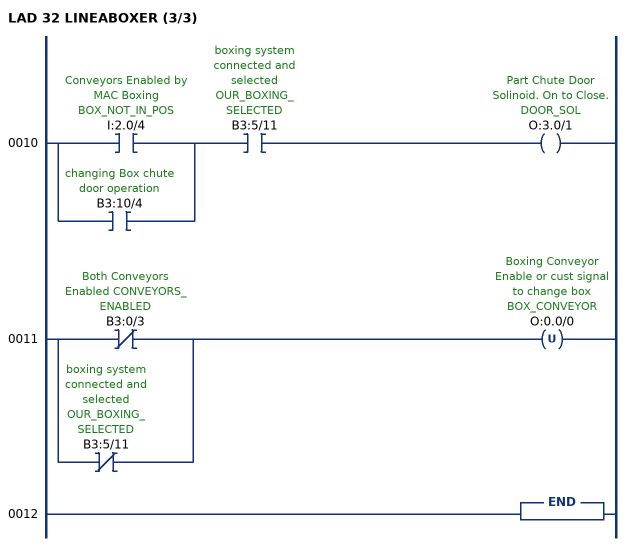
% Rung: 10 %
SOR BST XIC I:2.0/4 NXB XIC B3:10/4 BND XIC B3:5/11 OTE O:3.0/1 EOR
%   I:2.0/4  BOX_NOT_IN_POS  "Conveyors Enabled by MAC Boxing" %
%   B3:10/4  "changing Box chute door operation" %
%   B3:5/11  OUR_BOXING_SELECTED  "boxing system connected and selected" %
%   O:3.0/1  DOOR_SOL  "Part Chute Door Solinoid. On to Close." %
% Rung: 11 %
SOR BST XIO B3:0/3 NXB XIO B3:5/11 BND OTU O:0.0/0 EOR
%   B3:0/3  CONVEYORS_ENABLED  "Both Conveyors Enabled" %
%   B3:5/11  OUR_BOXING_SELECTED  "boxing system connected and selected" %
%   O:0.0/0  BOX_CONVEYOR  "Boxing Conveyor Enable or cust signal to change box" %
% Rung: 12 %
SOR END EOR

LADDER 33 "BULKBOXER"
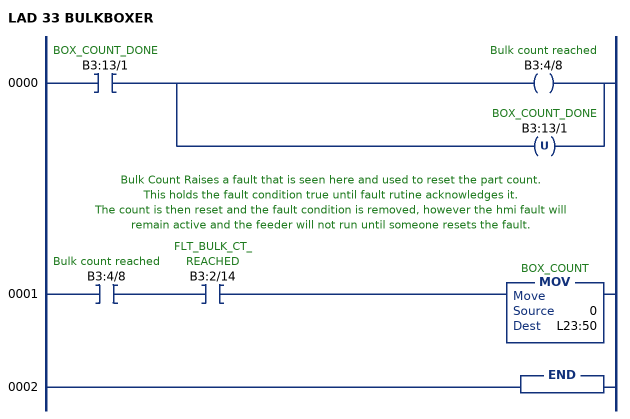
% Rung: 0 %
SOR XIC B3:13/1 BST OTE B3:4/8 NXB OTU B3:13/1 BND EOR
%   B3:13/1  BOX_COUNT_DONE %
%   B3:4/8  "Bulk count reached" %
% Rung: 1 %
% Bulk Count Raises a fault that is seen here and used to reset the part count.
% This holds the fault condition true until fault rutine acknowledges it.
% The count is then reset and the fault condition is removed, however the hmi fault will remain active and the feeder will not run until someone resets the fault. %
SOR XIC B3:4/8 XIC B3:2/14 MOV 0 L23:50 EOR
%   B3:4/8  "Bulk count reached" %
%   B3:2/14  FLT_BULK_CT_REACHED %
%   L23:50  BOX_COUNT %
% Rung: 2 %
SOR END EOR

LADDER 34 "CUSTBOXER"
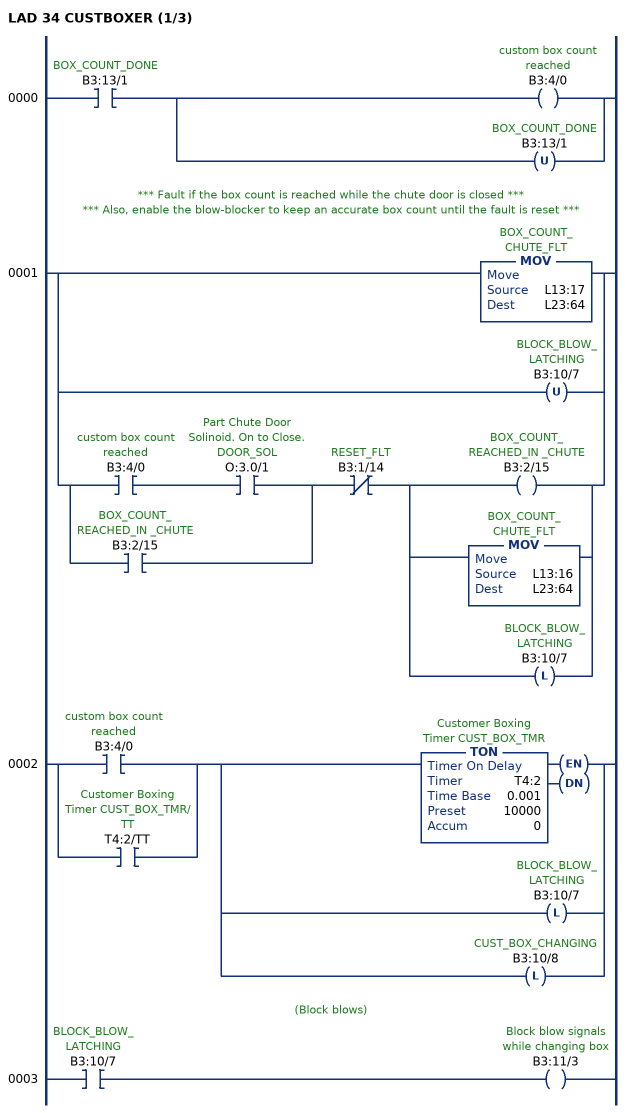
% Rung: 0 %
SOR XIC B3:13/1 BST OTE B3:4/0 NXB OTU B3:13/1 BND EOR
%   B3:13/1  BOX_COUNT_DONE %
%   B3:4/0  "custom box count reached" %
% Rung: 1 %
% *** Fault if the box count is reached while the chute door is closed ***
% *** Also, enable the blow-blocker to keep an accurate box count until the fault is reset *** %
SOR BST BST MOV L13:17 L23:64 NXB OTU B3:10/7 BND NXB BST XIC B3:4/0 XIC O:3.0/1 NXB XIC B3:2/15 BND XIO B3:1/14 BST OTE B3:2/15 NXB MOV L13:16 L23:64 NXB OTL B3:10/7 BND BND EOR
%   L13:17  FALSE %
%   L23:64  BOX_COUNT_CHUTE_FLT %
%   B3:10/7  BLOCK_BLOW_LATCHING %
%   B3:4/0  "custom box count reached" %
%   O:3.0/1  DOOR_SOL  "Part Chute Door Solinoid. On to Close." %
%   B3:2/15  "BOX_COUNT_REACHED_IN _CHUTE" %
%   B3:1/14  RESET_FLT %
%   L13:16  TRUE  "ONE TIME ENABLE FOR THE TIMES WHEN WE FORGET TO RE-ENABLE AFTER SHIPMENT" %
% Rung: 2 %
SOR BST XIC B3:4/0 NXB XIC T4:2/TT BND BST TON T4:2 0.001 10000 0 NXB OTL B3:10/7 NXB OTL B3:10/8 BND EOR
%   B3:4/0  "custom box count reached" %
%   T4:2  CUST_BOX_TMR  "Customer Boxing Timer" %
%   B3:10/7  BLOCK_BLOW_LATCHING %
%   B3:10/8  CUST_BOX_CHANGING %
% Rung: 3 %
% (Block blows) %
SOR XIC B3:10/7 OTE B3:11/3 EOR
%   B3:10/7  BLOCK_BLOW_LATCHING %
%   B3:11/3  "Block blow signals while changing box" %

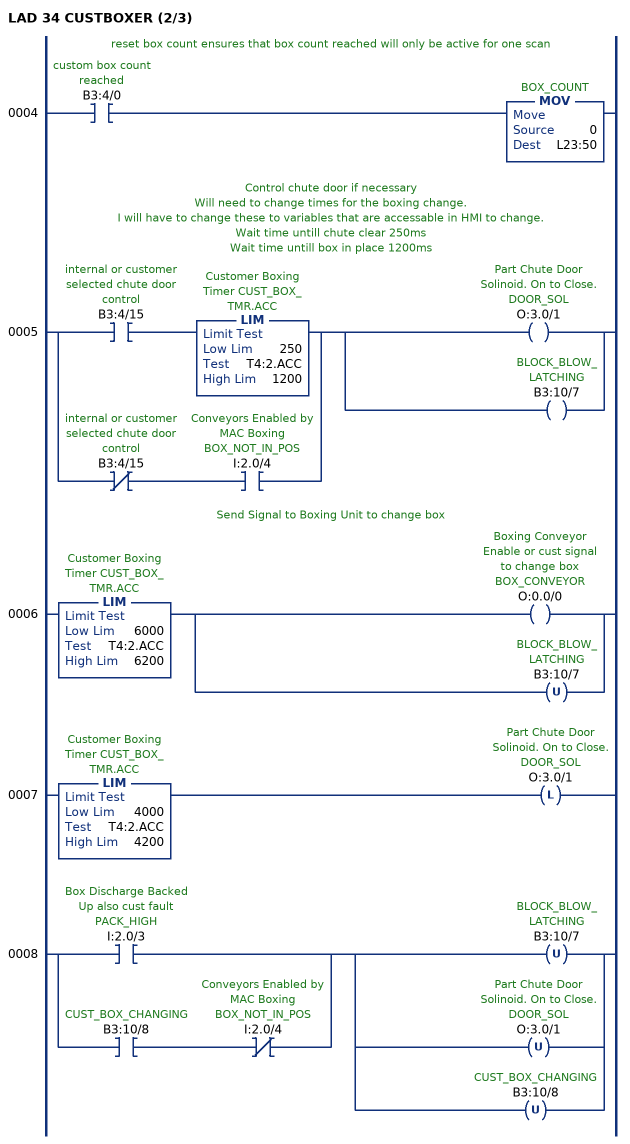
% Rung: 4 %
% reset box count ensures that box count reached will only be active for one scan %
SOR XIC B3:4/0 MOV 0 L23:50 EOR
%   B3:4/0  "custom box count reached" %
%   L23:50  BOX_COUNT %
% Rung: 5 %
% Control chute door if necessary
% 
% Will need to change times for the boxing change.
% I will have to change these to variables that are accessable in HMI to change.
% 
% Wait time untill chute clear 250ms
% Wait time untill box in place 1200ms %
SOR BST XIC B3:4/15 LIM 250 T4:2.ACC 1200 NXB XIO B3:4/15 XIC I:2.0/4 BND BST OTE O:3.0/1 NXB OTE B3:10/7 BND EOR
%   B3:4/15  "internal or customer selected chute door control" %
%   T4:2  CUST_BOX_TMR  "Customer Boxing Timer" %
%   I:2.0/4  BOX_NOT_IN_POS  "Conveyors Enabled by MAC Boxing" %
%   O:3.0/1  DOOR_SOL  "Part Chute Door Solinoid. On to Close." %
%   B3:10/7  BLOCK_BLOW_LATCHING %
% Rung: 6 %
% Send Signal to Boxing Unit to change box %
SOR LIM 6000 T4:2.ACC 6200 BST OTE O:0.0/0 NXB OTU B3:10/7 BND EOR
%   T4:2  CUST_BOX_TMR  "Customer Boxing Timer" %
%   O:0.0/0  BOX_CONVEYOR  "Boxing Conveyor Enable or cust signal to change box" %
%   B3:10/7  BLOCK_BLOW_LATCHING %
% Rung: 7 %
SOR LIM 4000 T4:2.ACC 4200 OTL O:3.0/1 EOR
%   T4:2  CUST_BOX_TMR  "Customer Boxing Timer" %
%   O:3.0/1  DOOR_SOL  "Part Chute Door Solinoid. On to Close." %
% Rung: 8 %
SOR BST XIC I:2.0/3 NXB XIC B3:10/8 XIO I:2.0/4 BND BST OTU B3:10/7 NXB OTU O:3.0/1 NXB OTU B3:10/8 BND EOR
%   I:2.0/3  PACK_HIGH  "Box Discharge Backed Up also cust fault" %
%   B3:10/8  CUST_BOX_CHANGING %
%   I:2.0/4  BOX_NOT_IN_POS  "Conveyors Enabled by MAC Boxing" %
%   B3:10/7  BLOCK_BLOW_LATCHING %
%   O:3.0/1  DOOR_SOL  "Part Chute Door Solinoid. On to Close." %

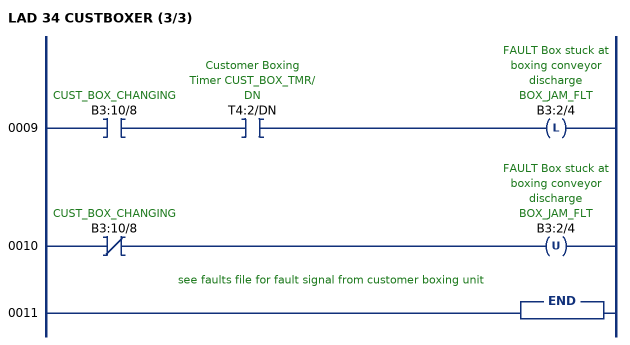
% Rung: 9 %
SOR XIC B3:10/8 XIC T4:2/DN OTL B3:2/4 EOR
%   B3:10/8  CUST_BOX_CHANGING %
%   T4:2  CUST_BOX_TMR  "Customer Boxing Timer" %
%   B3:2/4  BOX_JAM_FLT  "FAULT Box stuck at boxing conveyor discharge" %
% Rung: 10 %
SOR XIO B3:10/8 OTU B3:2/4 EOR
%   B3:10/8  CUST_BOX_CHANGING %
%   B3:2/4  BOX_JAM_FLT  "FAULT Box stuck at boxing conveyor discharge" %
% Rung: 11 %
% see faults file for fault signal from customer boxing unit %
SOR END EOR

LADDER 35 "CLEANUP"
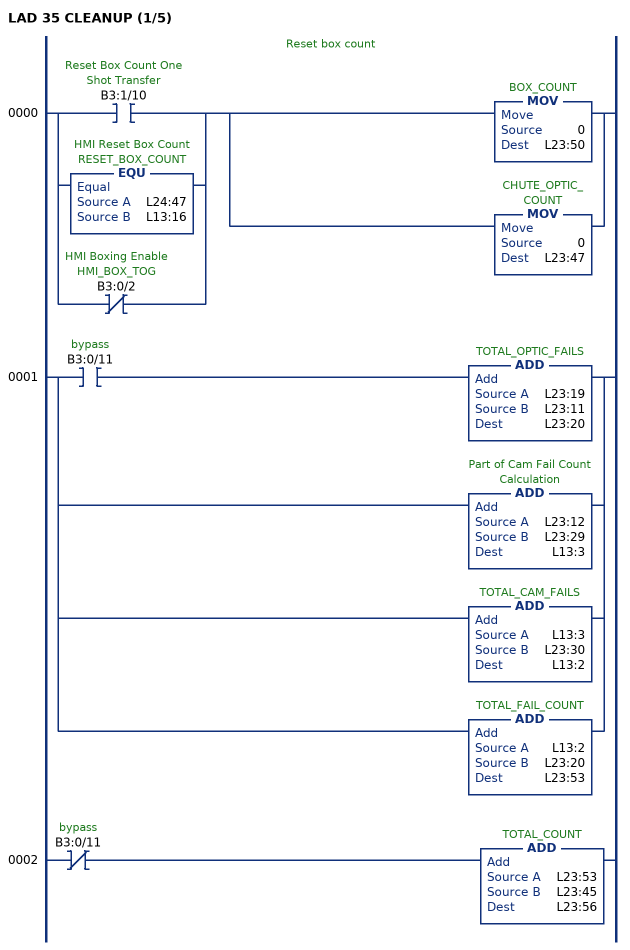
% Rung: 0 %
% Reset box count %
SOR BST XIC B3:1/10 NXB EQU L24:47 L13:16 NXB XIO B3:0/2 BND BST MOV 0 L23:50 NXB MOV 0 L23:47 BND EOR
%   B3:1/10  "Reset Box Count One Shot Transfer" %
%   L24:47  RESET_BOX_COUNT  "HMI Reset Box Count" %
%   L13:16  TRUE  "ONE TIME ENABLE FOR THE TIMES WHEN WE FORGET TO RE-ENABLE AFTER SHIPMENT" %
%   B3:0/2  HMI_BOX_TOG  "HMI Boxing Enable" %
%   L23:50  BOX_COUNT %
%   L23:47  CHUTE_OPTIC_COUNT %
% Rung: 1 %
SOR BST XIC B3:0/11 ADD L23:19 L23:11 L23:20 NXB ADD L23:12 L23:29 L13:3 NXB ADD L13:3 L23:30 L13:2 NXB ADD L13:2 L23:20 L23:53 BND EOR
%   B3:0/11  "bypass" %
%   L23:19  TOP_OPT_FAIL_CT %
%   L23:11  BOT_OPT_FAIL_CT %
%   L23:20  TOTAL_OPTIC_FAILS %
%   L23:12  BOT_NON_PASS  "parts missed BOT camera" %
%   L23:29  SIDE_NON_PASS  "parts missed side camera" %
%   L13:3  "Part of Cam Fail Count Calculation" %
%   L23:30  TOP_NON_PASS  "Parts Missed Top Camera" %
%   L13:2  TOTAL_CAM_FAILS %
%   L23:53  TOTAL_FAIL_COUNT %
% Rung: 2 %
SOR XIO B3:0/11 ADD L23:53 L23:45 L23:56 EOR
%   B3:0/11  "bypass" %
%   L23:53  TOTAL_FAIL_COUNT %
%   L23:45  BLOW_COUNT %
%   L23:56  TOTAL_COUNT %

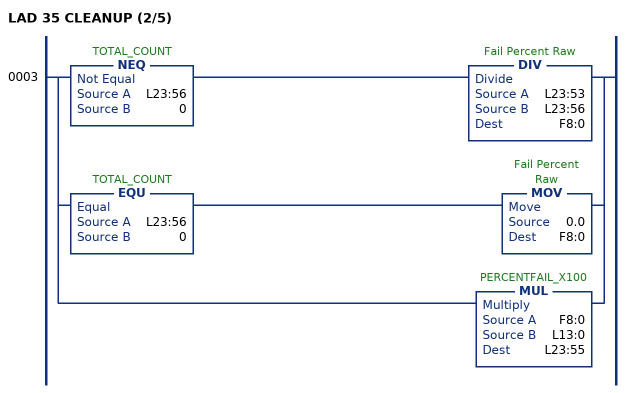
% Rung: 3 %
SOR BST NEQ L23:56 0 DIV L23:53 L23:56 F8:0 NXB EQU L23:56 0 MOV 0.0 F8:0 NXB MUL F8:0 L13:0 L23:55 BND EOR
%   L23:56  TOTAL_COUNT %
%   L23:53  TOTAL_FAIL_COUNT %
%   F8:0  "Fail Percent Raw" %
%   L13:0  "multiplyer to translate percent" %
%   L23:55  PERCENTFAIL_X100 %

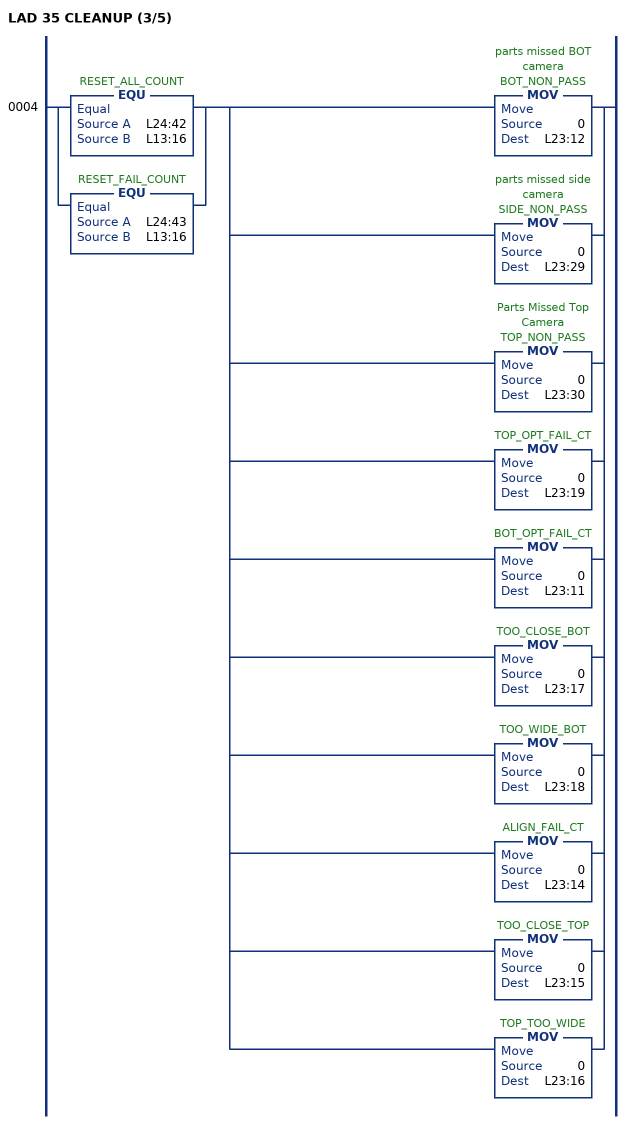
% Rung: 4 %
SOR BST EQU L24:42 L13:16 NXB EQU L24:43 L13:16 BND BST MOV 0 L23:12 NXB MOV 0 L23:29 NXB MOV 0 L23:30 NXB MOV 0 L23:19 NXB MOV 0 L23:11 NXB MOV 0 L23:17 NXB MOV 0 L23:18 NXB MOV 0 L23:14 NXB MOV 0 L23:15 NXB MOV 0 L23:16 BND EOR
%   L24:42  RESET_ALL_COUNT %
%   L13:16  TRUE  "ONE TIME ENABLE FOR THE TIMES WHEN WE FORGET TO RE-ENABLE AFTER SHIPMENT" %
%   L24:43  RESET_FAIL_COUNT %
%   L23:12  BOT_NON_PASS  "parts missed BOT camera" %
%   L23:29  SIDE_NON_PASS  "parts missed side camera" %
%   L23:30  TOP_NON_PASS  "Parts Missed Top Camera" %
%   L23:19  TOP_OPT_FAIL_CT %
%   L23:11  BOT_OPT_FAIL_CT %
%   L23:17  TOO_CLOSE_BOT %
%   L23:18  TOO_WIDE_BOT %
%   L23:14  ALIGN_FAIL_CT %
%   L23:15  TOO_CLOSE_TOP %
%   L23:16  TOP_TOO_WIDE %

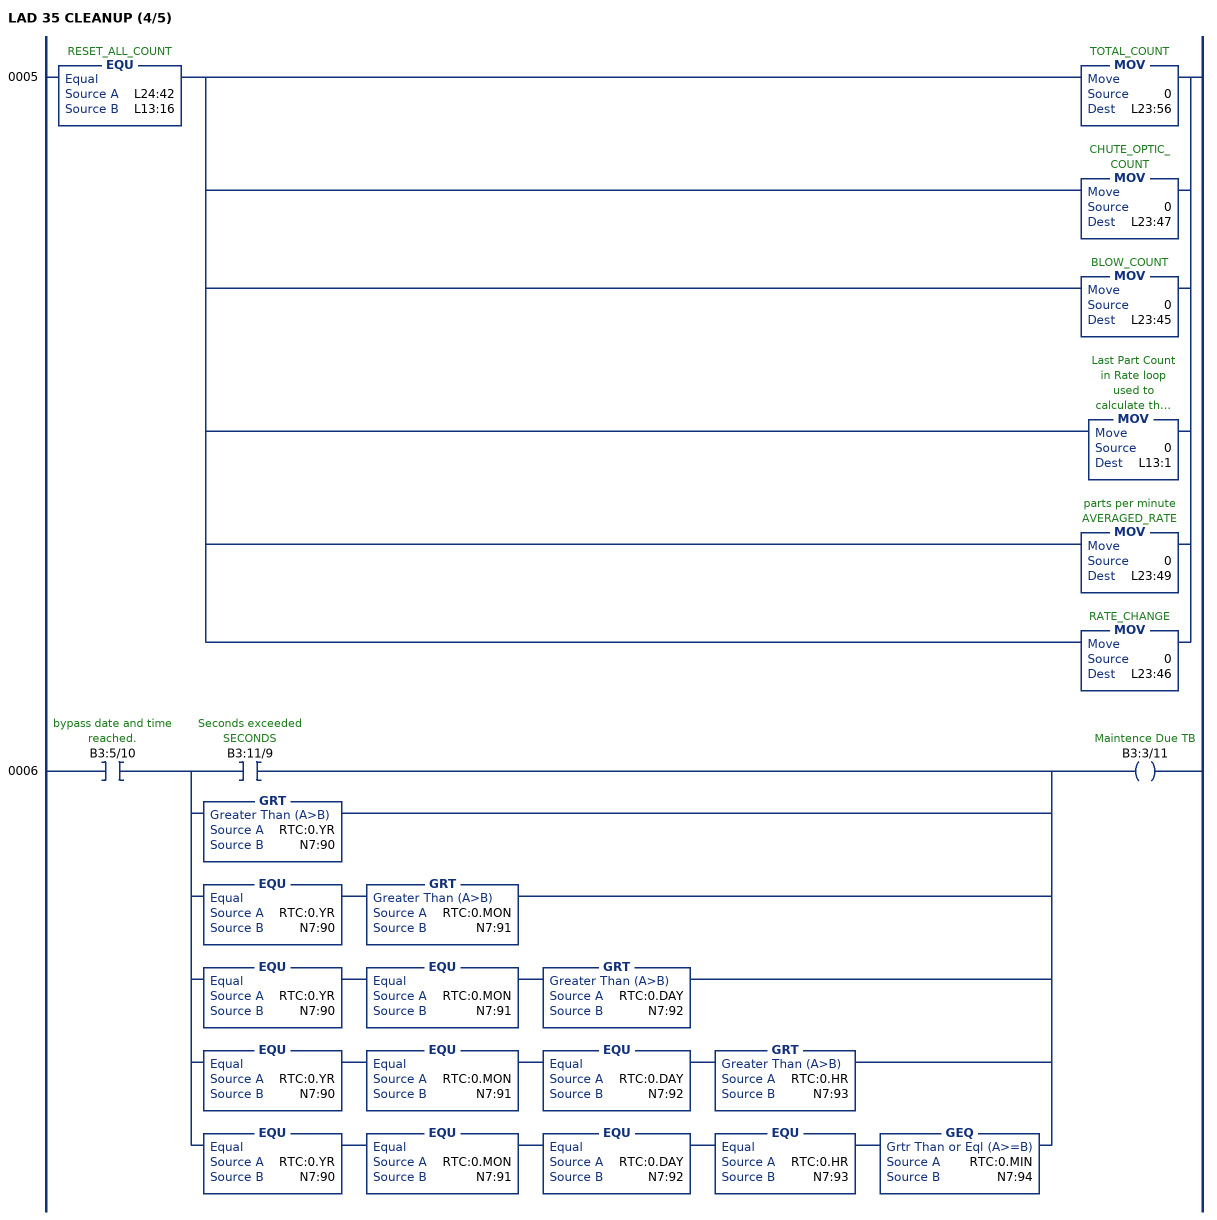
% Rung: 5 %
SOR EQU L24:42 L13:16 BST MOV 0 L23:56 NXB MOV 0 L23:47 NXB MOV 0 L23:45 NXB MOV 0 L13:1 NXB MOV 0 L23:49 NXB MOV 0 L23:46 BND EOR
%   L24:42  RESET_ALL_COUNT %
%   L13:16  TRUE  "ONE TIME ENABLE FOR THE TIMES WHEN WE FORGET TO RE-ENABLE AFTER SHIPMENT" %
%   L23:56  TOTAL_COUNT %
%   L23:47  CHUTE_OPTIC_COUNT %
%   L23:45  BLOW_COUNT %
%   L13:1  "Last Part Count in Rate loop used to calculate the last cycle part count" %
%   L23:49  AVERAGED_RATE  "parts per minute" %
%   L23:46  RATE_CHANGE %
% Rung: 6 %
SOR XIC B3:5/10 BST XIC B3:11/9 NXB GRT RTC:0.YR N7:90 NXB EQU RTC:0.YR N7:90 GRT RTC:0.MON N7:91 NXB EQU RTC:0.YR N7:90 EQU RTC:0.MON N7:91 GRT RTC:0.DAY N7:92 NXB EQU RTC:0.YR N7:90 EQU RTC:0.MON N7:91 EQU RTC:0.DAY N7:92 GRT RTC:0.HR N7:93 NXB EQU RTC:0.YR N7:90 EQU RTC:0.MON N7:91 EQU RTC:0.DAY N7:92 EQU RTC:0.HR N7:93 GEQ RTC:0.MIN N7:94 BND OTE B3:3/11 EOR
%   B3:5/10  "bypass date and time reached." %
%   B3:11/9  SECONDS  "Seconds exceeded" %
%   N7:90  RTC %
%   B3:3/11  TB  "Maintence Due" %

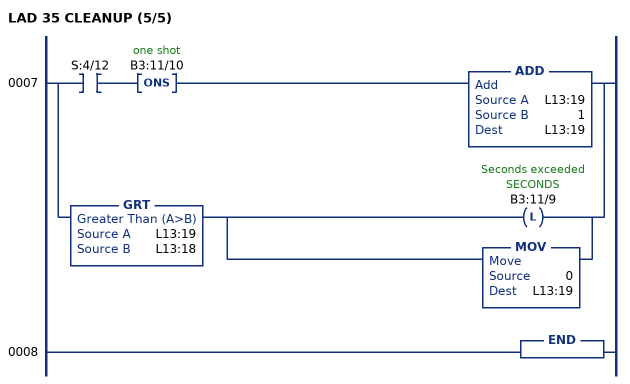
% Rung: 7 %
SOR BST XIC S:4/12 ONS B3:11/10 ADD L13:19 1 L13:19 NXB GRT L13:19 L13:18 BST OTL B3:11/9 NXB MOV 0 L13:19 BND BND EOR
%   B3:11/10  "one shot" %
%   L13:18  MAX %
%   B3:11/9  SECONDS  "Seconds exceeded" %
% Rung: 8 %
SOR END EOR

LADDER 36 "J_CUST_BOX"    % Justin's customer boxing ladder %
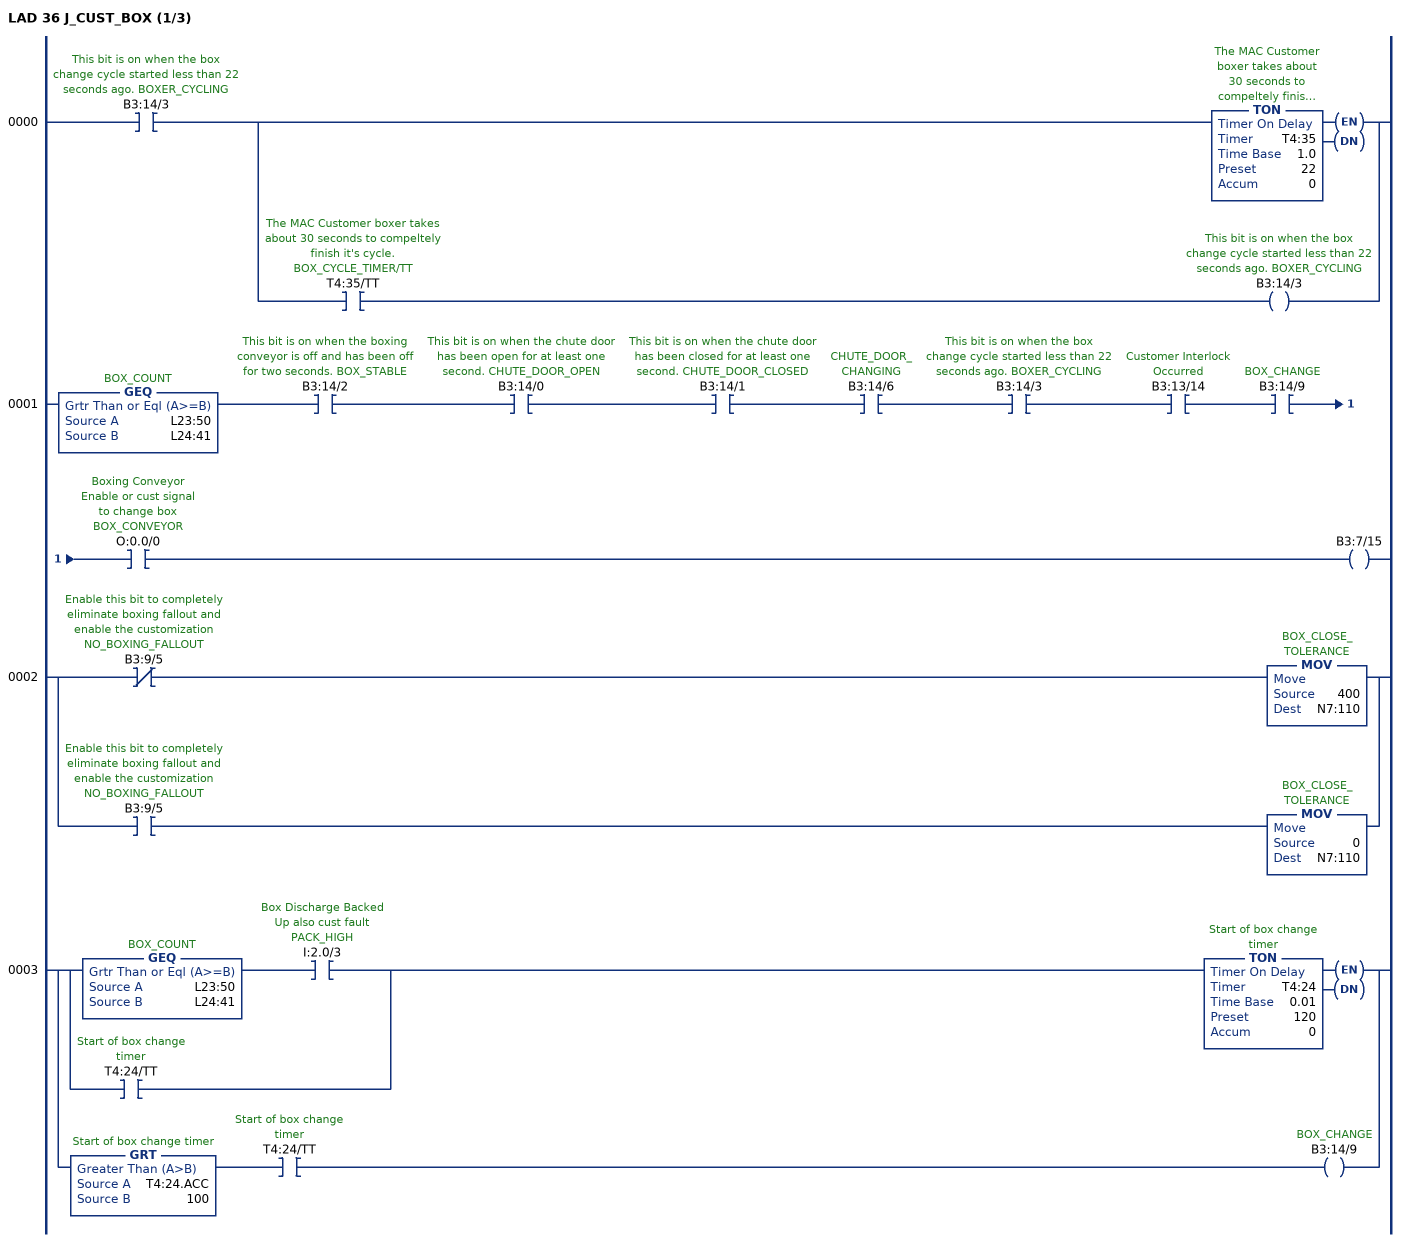
% Rung: 0 %
SOR XIC B3:14/3 BST TON T4:35 1.0 22 0 NXB XIC T4:35/TT OTE B3:14/3 BND EOR
%   B3:14/3  BOXER_CYCLING  "This bit is on when the box change cycle started less than 22 seconds ago." %
%   T4:35  BOX_CYCLE_TIMER  "The MAC Customer boxer takes about 30 seconds to compeltely finish it's cycle." %
% Rung: 1 %
SOR GEQ L23:50 L24:41 XIC B3:14/2 XIC B3:14/0 XIC B3:14/1 XIC B3:14/6 XIC B3:14/3 XIC B3:13/14 XIC B3:14/9 XIC O:0.0/0 OTE B3:7/15 EOR
%   L23:50  BOX_COUNT %
%   L24:41  BOX_COUNT_LIMIT %
%   B3:14/2  BOX_STABLE  "This bit is on when the boxing conveyor is off and has been off for two seconds." %
%   B3:14/0  CHUTE_DOOR_OPEN  "This bit is on when the chute door has been open for at least one second." %
%   B3:14/1  CHUTE_DOOR_CLOSED  "This bit is on when the chute door has been closed for at least one second." %
%   B3:14/6  CHUTE_DOOR_CHANGING %
%   B3:14/3  BOXER_CYCLING  "This bit is on when the box change cycle started less than 22 seconds ago." %
%   B3:13/14  "Customer Interlock Occurred" %
%   B3:14/9  BOX_CHANGE %
%   O:0.0/0  BOX_CONVEYOR  "Boxing Conveyor Enable or cust signal to change box" %
% Rung: 2 %
SOR BST XIO B3:9/5 MOV 400 N7:110 NXB XIC B3:9/5 MOV 0 N7:110 BND EOR
%   B3:9/5  NO_BOXING_FALLOUT  "Enable this bit to completely eliminate boxing fallout and enable the customization" %
%   N7:110  BOX_CLOSE_TOLERANCE %
% Rung: 3 %
SOR BST BST GEQ L23:50 L24:41 XIC I:2.0/3 NXB XIC T4:24/TT BND TON T4:24 0.01 120 0 NXB GRT T4:24.ACC 100 XIC T4:24/TT OTE B3:14/9 BND EOR
%   L23:50  BOX_COUNT %
%   L24:41  BOX_COUNT_LIMIT %
%   I:2.0/3  PACK_HIGH  "Box Discharge Backed Up also cust fault" %
%   T4:24  "Start of box change timer" %
%   B3:14/9  BOX_CHANGE %

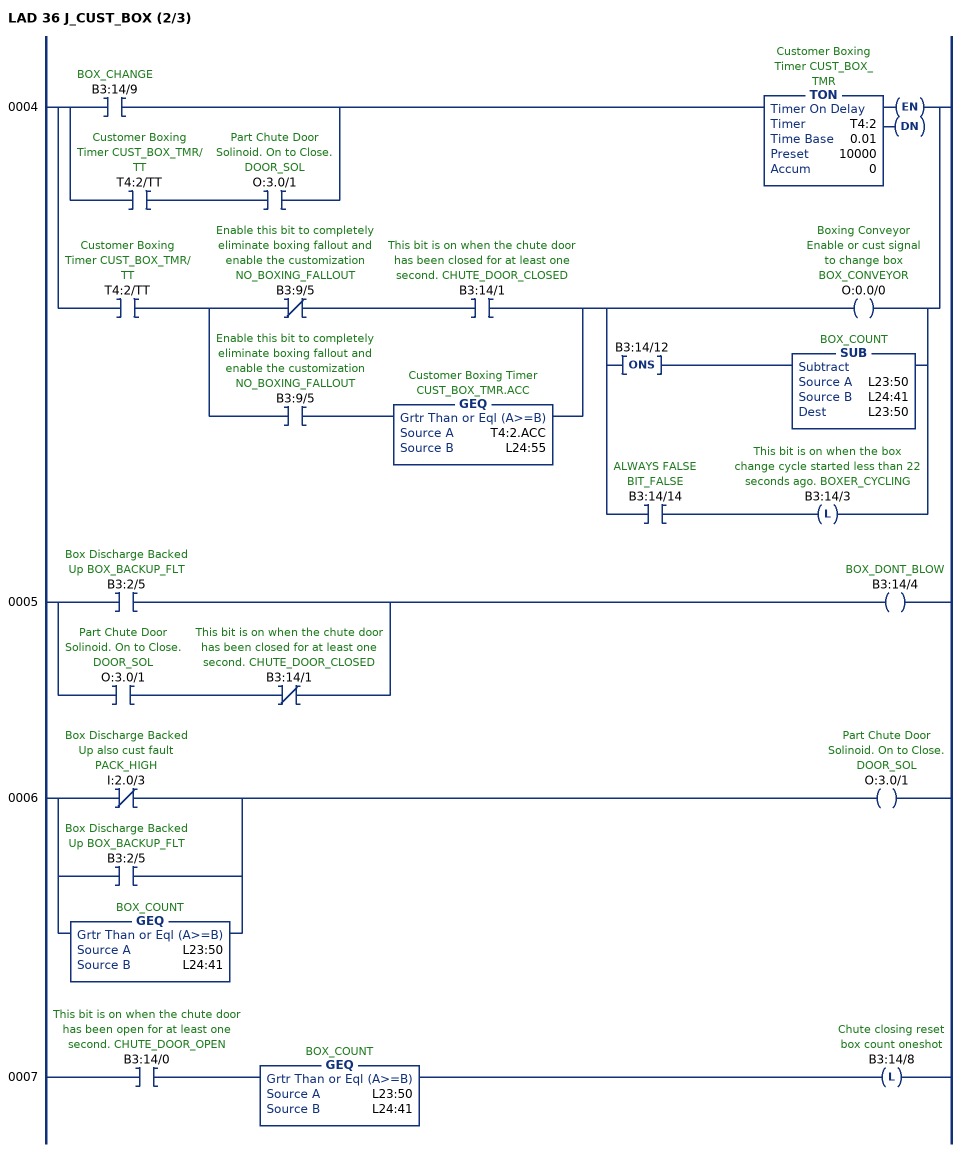
% Rung: 4 %
SOR BST BST XIC B3:14/9 NXB XIC T4:2/TT XIC O:3.0/1 BND TON T4:2 0.01 10000 0 NXB XIC T4:2/TT BST XIO B3:9/5 XIC B3:14/1 NXB XIC B3:9/5 GEQ T4:2.ACC L24:55 BND BST OTE O:0.0/0 NXB ONS B3:14/12 SUB L23:50 L24:41 L23:50 NXB XIC B3:14/14 OTL B3:14/3 BND BND EOR
%   B3:14/9  BOX_CHANGE %
%   T4:2  CUST_BOX_TMR  "Customer Boxing Timer" %
%   O:3.0/1  DOOR_SOL  "Part Chute Door Solinoid. On to Close." %
%   B3:9/5  NO_BOXING_FALLOUT  "Enable this bit to completely eliminate boxing fallout and enable the customization" %
%   B3:14/1  CHUTE_DOOR_CLOSED  "This bit is on when the chute door has been closed for at least one second." %
%   L24:55  CHUTE_CLOSE_DELAY  "Timer to allow parts to pass through the chute" %
%   O:0.0/0  BOX_CONVEYOR  "Boxing Conveyor Enable or cust signal to change box" %
%   L23:50  BOX_COUNT %
%   L24:41  BOX_COUNT_LIMIT %
%   B3:14/14  BIT_FALSE  "ALWAYS FALSE" %
%   B3:14/3  BOXER_CYCLING  "This bit is on when the box change cycle started less than 22 seconds ago." %
% Rung: 5 %
SOR BST XIC B3:2/5 NXB XIC O:3.0/1 XIO B3:14/1 BND OTE B3:14/4 EOR
%   B3:2/5  BOX_BACKUP_FLT  "Box Discharge Backed Up" %
%   O:3.0/1  DOOR_SOL  "Part Chute Door Solinoid. On to Close." %
%   B3:14/1  CHUTE_DOOR_CLOSED  "This bit is on when the chute door has been closed for at least one second." %
%   B3:14/4  BOX_DONT_BLOW %
% Rung: 6 %
SOR BST XIO I:2.0/3 NXB XIC B3:2/5 NXB GEQ L23:50 L24:41 BND OTE O:3.0/1 EOR
%   I:2.0/3  PACK_HIGH  "Box Discharge Backed Up also cust fault" %
%   B3:2/5  BOX_BACKUP_FLT  "Box Discharge Backed Up" %
%   L23:50  BOX_COUNT %
%   L24:41  BOX_COUNT_LIMIT %
%   O:3.0/1  DOOR_SOL  "Part Chute Door Solinoid. On to Close." %
% Rung: 7 %
SOR XIC B3:14/0 GEQ L23:50 L24:41 OTL B3:14/8 EOR
%   B3:14/0  CHUTE_DOOR_OPEN  "This bit is on when the chute door has been open for at least one second." %
%   L23:50  BOX_COUNT %
%   L24:41  BOX_COUNT_LIMIT %
%   B3:14/8  "Chute closing reset box count oneshot" %

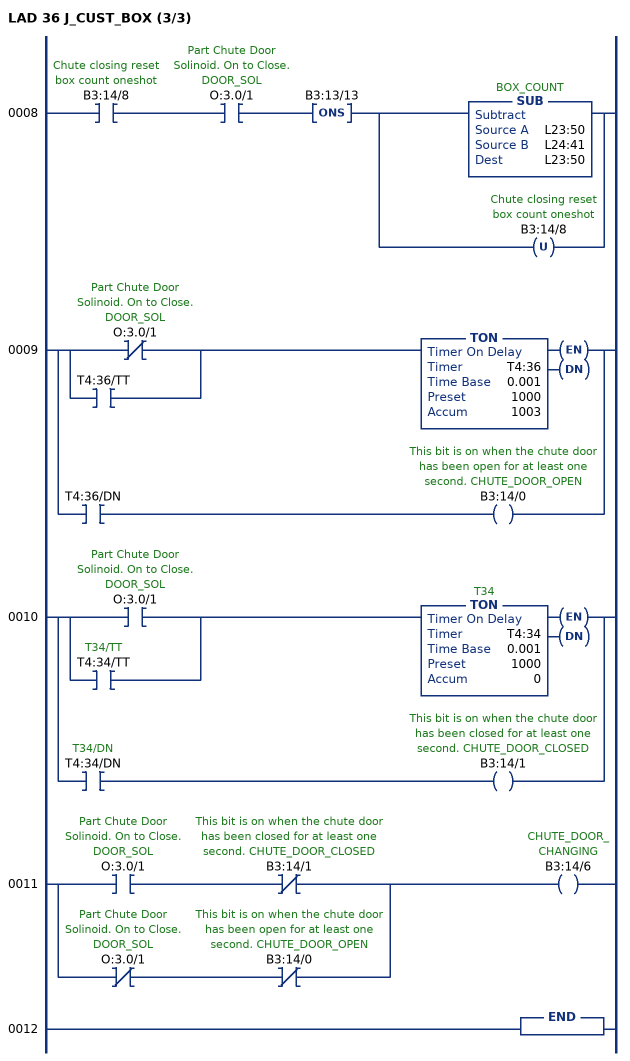
% Rung: 8 %
SOR XIC B3:14/8 XIC O:3.0/1 ONS B3:13/13 BST SUB L23:50 L24:41 L23:50 NXB OTU B3:14/8 BND EOR
%   B3:14/8  "Chute closing reset box count oneshot" %
%   O:3.0/1  DOOR_SOL  "Part Chute Door Solinoid. On to Close." %
%   L23:50  BOX_COUNT %
%   L24:41  BOX_COUNT_LIMIT %
% Rung: 9 %
SOR BST BST XIO O:3.0/1 NXB XIC T4:36/TT BND TON T4:36 0.001 1000 1003 NXB XIC T4:36/DN OTE B3:14/0 BND EOR
%   O:3.0/1  DOOR_SOL  "Part Chute Door Solinoid. On to Close." %
%   B3:14/0  CHUTE_DOOR_OPEN  "This bit is on when the chute door has been open for at least one second." %
% Rung: 10 %
SOR BST BST XIC O:3.0/1 NXB XIC T4:34/TT BND TON T4:34 0.001 1000 0 NXB XIC T4:34/DN OTE B3:14/1 BND EOR
%   O:3.0/1  DOOR_SOL  "Part Chute Door Solinoid. On to Close." %
%   T4:34  T34 %
%   B3:14/1  CHUTE_DOOR_CLOSED  "This bit is on when the chute door has been closed for at least one second." %
% Rung: 11 %
SOR BST XIC O:3.0/1 XIO B3:14/1 NXB XIO O:3.0/1 XIO B3:14/0 BND OTE B3:14/6 EOR
%   O:3.0/1  DOOR_SOL  "Part Chute Door Solinoid. On to Close." %
%   B3:14/1  CHUTE_DOOR_CLOSED  "This bit is on when the chute door has been closed for at least one second." %
%   B3:14/0  CHUTE_DOOR_OPEN  "This bit is on when the chute door has been open for at least one second." %
%   B3:14/6  CHUTE_DOOR_CHANGING %
% Rung: 12 %
SOR END EOR

LADDER 37 "BOXING"
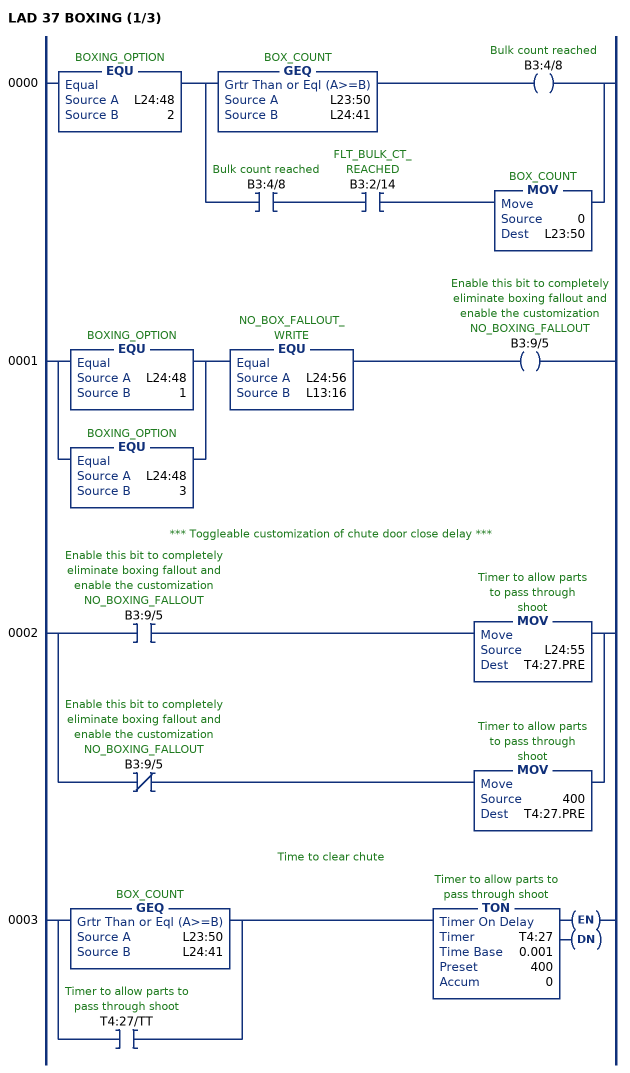
% Rung: 0 %
SOR EQU L24:48 2 BST GEQ L23:50 L24:41 OTE B3:4/8 NXB XIC B3:4/8 XIC B3:2/14 MOV 0 L23:50 BND EOR
%   L24:48  BOXING_OPTION %
%   L23:50  BOX_COUNT %
%   L24:41  BOX_COUNT_LIMIT %
%   B3:4/8  "Bulk count reached" %
%   B3:2/14  FLT_BULK_CT_REACHED %
% Rung: 1 %
SOR BST EQU L24:48 1 NXB EQU L24:48 3 BND EQU L24:56 L13:16 OTE B3:9/5 EOR
%   L24:48  BOXING_OPTION %
%   L24:56  NO_BOX_FALLOUT_WRITE %
%   L13:16  TRUE  "ONE TIME ENABLE FOR THE TIMES WHEN WE FORGET TO RE-ENABLE AFTER SHIPMENT" %
%   B3:9/5  NO_BOXING_FALLOUT  "Enable this bit to completely eliminate boxing fallout and enable the customization" %
% Rung: 2 %
% *** Toggleable customization of chute door close delay *** %
SOR BST XIC B3:9/5 MOV L24:55 T4:27.PRE NXB XIO B3:9/5 MOV 400 T4:27.PRE BND EOR
%   B3:9/5  NO_BOXING_FALLOUT  "Enable this bit to completely eliminate boxing fallout and enable the customization" %
%   L24:55  CHUTE_CLOSE_DELAY  "Timer to allow parts to pass through the chute" %
%   T4:27  "Timer to allow parts to pass through shoot" %
% Rung: 3 %
% Time to clear chute %
SOR BST GEQ L23:50 L24:41 NXB XIC T4:27/TT BND TON T4:27 0.001 400 0 EOR
%   L23:50  BOX_COUNT %
%   L24:41  BOX_COUNT_LIMIT %
%   T4:27  "Timer to allow parts to pass through shoot" %

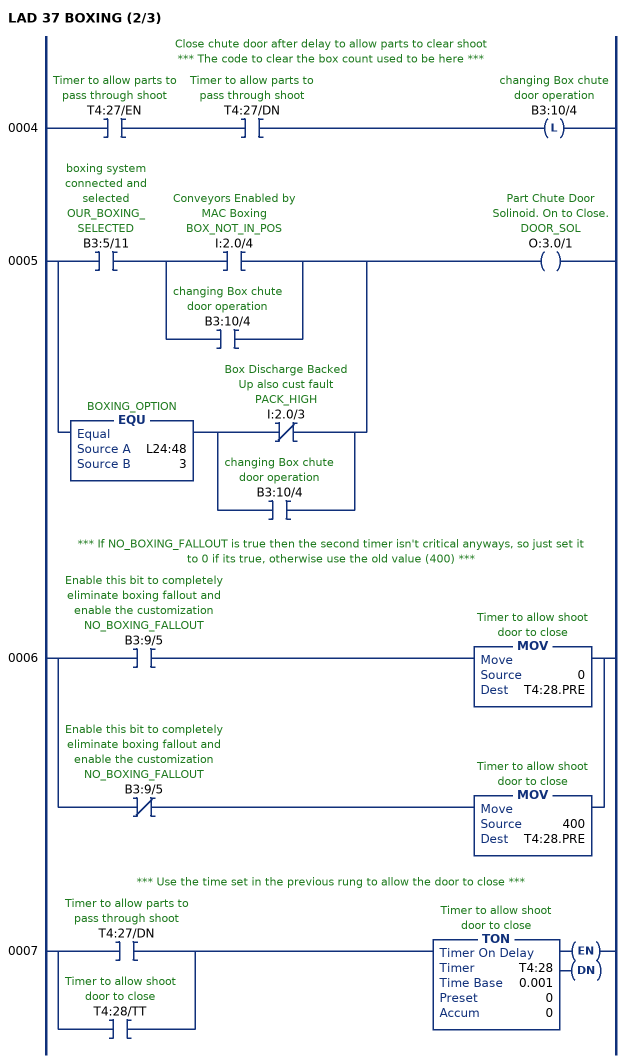
% Rung: 4 %
% Close chute door after delay to allow parts to clear shoot
% *** The code to clear the box count used to be here *** %
SOR XIC T4:27/EN XIC T4:27/DN OTL B3:10/4 EOR
%   T4:27  "Timer to allow parts to pass through shoot" %
%   B3:10/4  "changing Box chute door operation" %
% Rung: 5 %
SOR BST XIC B3:5/11 BST XIC I:2.0/4 NXB XIC B3:10/4 BND NXB EQU L24:48 3 BST XIO I:2.0/3 NXB XIC B3:10/4 BND BND OTE O:3.0/1 EOR
%   B3:5/11  OUR_BOXING_SELECTED  "boxing system connected and selected" %
%   I:2.0/4  BOX_NOT_IN_POS  "Conveyors Enabled by MAC Boxing" %
%   B3:10/4  "changing Box chute door operation" %
%   L24:48  BOXING_OPTION %
%   I:2.0/3  PACK_HIGH  "Box Discharge Backed Up also cust fault" %
%   O:3.0/1  DOOR_SOL  "Part Chute Door Solinoid. On to Close." %
% Rung: 6 %
% *** If NO_BOXING_FALLOUT is true then the second timer isn't critical anyways, so just set it to 0 if its true, otherwise use the old value (400) *** %
SOR BST XIC B3:9/5 MOV 0 T4:28.PRE NXB XIO B3:9/5 MOV 400 T4:28.PRE BND EOR
%   B3:9/5  NO_BOXING_FALLOUT  "Enable this bit to completely eliminate boxing fallout and enable the customization" %
%   T4:28  "Timer to allow shoot door to close" %
% Rung: 7 %
% *** Use the time set in the previous rung to allow the door to close *** %
SOR BST XIC T4:27/DN NXB XIC T4:28/TT BND TON T4:28 0.001 0 0 EOR
%   T4:27  "Timer to allow parts to pass through shoot" %
%   T4:28  "Timer to allow shoot door to close" %

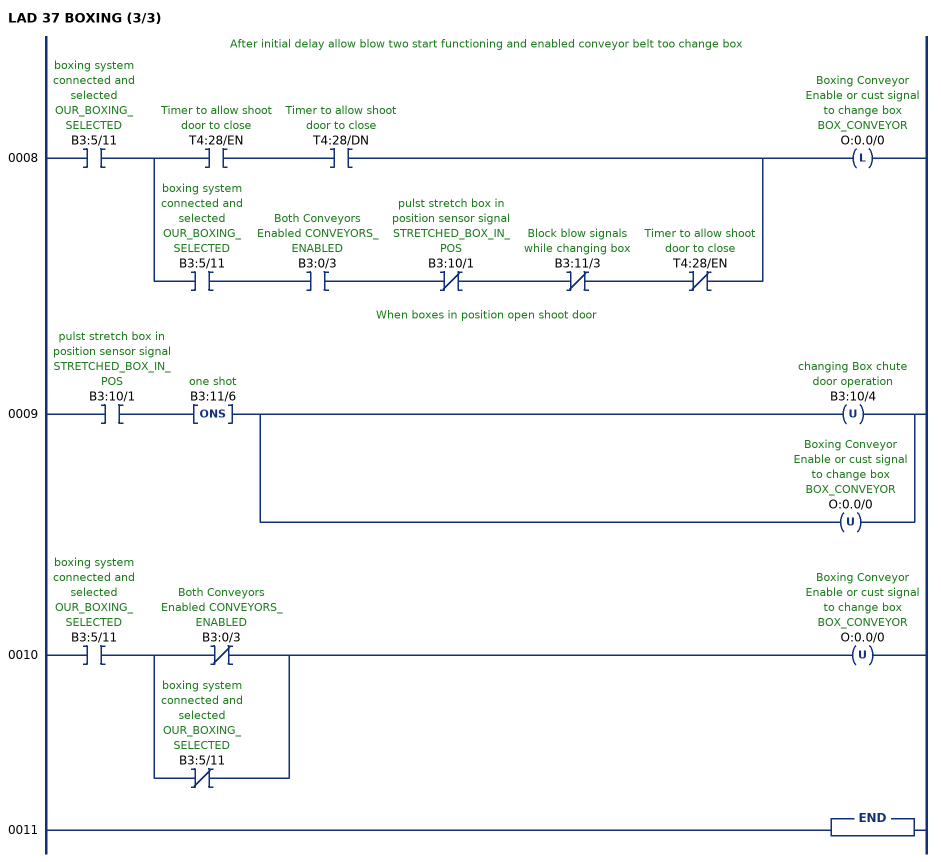
% Rung: 8 %
% After initial delay allow blow two start functioning and enabled conveyor belt too change box %
SOR XIC B3:5/11 BST XIC T4:28/EN XIC T4:28/DN NXB XIC B3:5/11 XIC B3:0/3 XIO B3:10/1 XIO B3:11/3 XIO T4:28/EN BND OTL O:0.0/0 EOR
%   B3:5/11  OUR_BOXING_SELECTED  "boxing system connected and selected" %
%   T4:28  "Timer to allow shoot door to close" %
%   B3:0/3  CONVEYORS_ENABLED  "Both Conveyors Enabled" %
%   B3:10/1  STRETCHED_BOX_IN_POS  "pulst stretch box in position sensor signal" %
%   B3:11/3  "Block blow signals while changing box" %
%   O:0.0/0  BOX_CONVEYOR  "Boxing Conveyor Enable or cust signal to change box" %
% Rung: 9 %
% When boxes in position open shoot door %
SOR XIC B3:10/1 ONS B3:11/6 BST OTU B3:10/4 NXB OTU O:0.0/0 BND EOR
%   B3:10/1  STRETCHED_BOX_IN_POS  "pulst stretch box in position sensor signal" %
%   B3:11/6  "one shot" %
%   B3:10/4  "changing Box chute door operation" %
%   O:0.0/0  BOX_CONVEYOR  "Boxing Conveyor Enable or cust signal to change box" %
% Rung: 10 %
SOR XIC B3:5/11 BST XIO B3:0/3 NXB XIO B3:5/11 BND OTU O:0.0/0 EOR
%   B3:5/11  OUR_BOXING_SELECTED  "boxing system connected and selected" %
%   B3:0/3  CONVEYORS_ENABLED  "Both Conveyors Enabled" %
%   O:0.0/0  BOX_CONVEYOR  "Boxing Conveyor Enable or cust signal to change box" %
% Rung: 11 %
SOR END EOR

OTHER DOCUMENTED ADDRESSES
  100000L  
  B3:2/12  "Rate Drop Fault Possible Feed Jam"
  B3:5/8  OFF
  B3:5/13  "bot result toggle"
  B3:6/5  "bottom top camra pass zone"
  B3:6/6  "one shot"
  B3:6/7  EI3_OLD  "Enable Inspection 3"
  B3:6/9  CONV_ON  "both conveyors enabled"
  B3:6/10  "Bypass un-needed code untill completed !!!!!!!!!!!!!!!!"
  B3:6/15  "nothing"
  B3:7/2  "bypass"
  B3:7/5  "extra bypass"
  B3:7/8  "top camera pass part zone"
  B3:7/11  "good part detected at top top"
  B3:7/12  "side camera pass part zone"
  B3:7/14  "passing part present bottom top camera"
  B3:8/0  "bypass extra trigger camera 1"
  B3:8/1  "bypass extra trigger camera 2"
  B3:8/2  "bypass extra trigger camera 3"
  B3:8/3  "bypass extra trigger camera 4"
  B3:8/5  TEST  "FORCE FEED ON/OFF"
  B3:8/6  "a bypass bit"
  B3:8/7  "a bypass bit"
  B3:8/11  ET4  "extra trigger camera 4"
  B3:8/12  "start bottom top camera responce"
  B3:8/13  "extra blow signal for testing"
  B3:8/15  "start side camera responce"
  B3:9/2  "one shot"
  B3:9/4  "start top camera responce"
  B3:9/7  "C1t"
  B3:9/8  "C2D"
  B3:9/9  "C2t"
  B3:9/14  "input from hmi to reset count"
  B3:10/0  "bypass part too close"
  B3:10/5  "one shot"
  B3:10/6  "excessive data output time"
  B3:10/9  "one shot"
  B3:10/10  "one shot"
  B3:10/14  "Dont use"
  B3:11/0  "bypass unused portion of code"
  B3:11/1  "bypass"
  B3:11/2  "Enable encoder belt movement simulation when testing"
  B3:11/7  "one shot"
  B3:11/11  "one shot"
  B3:11/13  TEST_TRIG_SIG
  B3:11/14  SOC  "start delay to false optic cycle"
  B3:11/15  "one shot"
  B3:12/2  "Command 2 Oneshot"
  B3:12/3  "Command 2 Active"
  B3:12/4  "Command3 Oneshot"
  B3:12/5  "Command 3 Active"
  B3:12/6  "Inspection Command Counter"
  B3:12/7  "Command 4 Active"
  B3:12/8  "Command 4 Oneshot"
  B3:12/15  "FALSE"
  B3:13/5  "bypass"
  B3:13/12  "Test Trigger to laser Spacing"
  B3:13/15  "Test Signals"
  B3:14  BOXING_STATUS  "Various bits all used in boxing"
  B3:14/5  BOX_CLOSE_CHUTE
  B3:14/7  CHUTE_CLOSE
  B3:17/12  "Always Off"
  B9:0/0  "Trigger Insert Position"
  B9:0/1  "bottom of top conveyor part transfer location"
  B9:0/[N7:2]  "Mask Start Position"
  B9:0/[N7:6]  "Blow Off Position"
  B9:0/[N7:20]  "part present bit shift load position"
  B9:0/[N16:0]  "Trigger Position"
  B9:0/[N17:8]  "part from bottom belt present at top belt optic position"
  B10:0/0  "Pass Insert Position"
  B10:0/1  TOP_CAM_LOAD
  B10:0/[N7:2]  "Pass Bit Position"
  B10:0/[N7:4]  "Pass Insert Position"
  B10:0/[N7:5]  "Pass Start Position"
  B10:0/[N7:6]  "Pass Position"
  B10:0/[N7:48]  TOPCAMTRIGPOS
  B10:0/[N16:4]  "Pass Insert Position"
  B10:0/[N16:6]  "Pass Position"
  B11:0/0  "Trigger Insert Position"
  B11:0/[N7:8]  "Fail Bit Position"
  B11:0/[N7:28]  "Bot Camera Trigger Posistion"
  B11:0/[N16:0]  "Trigger Position"
  B12:1/0  "Conveyor Start Oneshot"
  B12:1/1  "Feed Start Oneshot"
  B12:1/2  "Conveyor Stop Oneshot"
  B12:1/3  "Feed Stop Oneshot"
  B12:1/5  "Conveyor Start Oneshot"
  B12:2/8  BOXING  "BOXING System Wiring Is Connected"
  B12:2/10  OSR_42
  B12:2/11  BOX_IN_POS_OS  "BOXING Empty Box In Position One-Shot"
  B12:2/12  BOX_INDEXING  "BOXING Conveyor Indexing"
  B12:2/13  OSR_45
  B12:2/14  BOX_PLC_COUNTER  "BOXING PLC Counter Active Bit"
  B14:0/0  "Bottom Pass Insert"
  B14:0/4  "Bottom Pass Insert Position"
  B14:0/[N13:14]  "Start Laser Pass"
  B14:0/[N16:4]  "Pass Insert Position"
  B14:0/[N16:6]  "Pass Position"
  B15:0  "Alarm Bits"
  B18:1/1  "bottom pass one shot transfer"
  B18:3/2  "Part Present Oneshot"
  B18:3/3  "Part Present Oneshot"
  B18:5/11  "Transfer bottom pass result from end of bottom conveyor"
  B18:10/15  "Reserved For Shift Registers"
  B18:142  "fack camerea pass signal"
  B22:0  "Transfer Shift Register"
  B22:0/0  "load top conveyor bitshift from bottom cammera pass."
  B22:0/[N17:8]  "bottom good part at top optic position"
  B23:0/[N7:0]  "Bottom Pass Output"
  B25:0/4  UNUSED_4  "Unused Camera #4 Trigger"
  BOTTOM_CONVEYOR  
  BOX_CYCLING  
  C5:2  "Fault Counter"
  C5:5  "Trigger Count"
  C5:6  "Trigger Counter"
  C5:7  "Complete Counter"
  C5:8  BOX_CNT_1  "BOXING Quantity Counter #1"
  C5:9  BOX_CNT_2  "BOXING Quantity Counter #1"
  CHUTE_OPC  
  ENABLE_I1  "ENABLE_I1"
  F8:5  "bottom top camera pass count"
  F8:6  "top top camera missed count"
  F8:7  "top side camera missed count"
  F8:8  "bot top camera missed part count"
  F8:26  "Part bits loaded into BitShift"
  F8:29  "Count of signals passed to the blow valve"
  F8:30  BOT_NON_PASS_OLD  "Parts missed bot camera"
  F8:31  "Count of off alignment between top and bottom ALIGN_FAILS"
  F8:33  TOP_NON_PASS_OLD  "parts missed top camera"
  F8:34  "count of blow signals"
  F8:35  "rate difference"
  F8:36  2MIN_OF_RATE  "OLD AND NEW ADDED TOGETHER"
  F8:38  "averaged rate"
  F8:39  SIDE_NON_PASS_OLD  "parts missed side camera"
  F8:42  "Total fail and missed count CAM_NON_PASS"
  F8:43  "change in part rate as %"
  F8:44  "difference as a ratio of the total"
  F8:45  "TOO_CLOSE_BOT"
  F8:46  "TOO_WIDE_BOT"
  F8:48  "transfer"
  F8:49  "TOO_CLOSE_TOP"
  F8:51  "TOO_WIDE_TOP"
  F8:52  "OPTO_FAILS"
  F8:53  "optic fail count top camera TOP_OPT_FAIL_CT"
  F8:54  "optic fail count bot camera BOT_OPT_FAIL_CT"
  F19:0  BOT_HS_COUNTER  "Bottom Encoder High Speed Counter"
  F19:4  "Conveyor Input Blip Counter"
  HSC:0  "top conveyor"
  HSC:0.3/6  "Underflow interrupt"
  HSC:0.3/7  "Overflow interrupt"
  HSC:1  "bottom conveyor"
  HSC:1.3/6  "Underflow interrupt"
  HSC:1.3/7  "Overflow interrupt"
  I:0.0/0  "Bottom Conveyor Encoder Signal "A""
  I:0.0/1  "Bottom Conveyor Encoder Signal "B""
  I:0.0/4  "Top Conveyor Encoder Signal "A""
  I:0.0/5  "Top Conveyor Encoder Signal "B""
  I:0.2/3  "Packaging Conveyor full"
  I:0.2/4  "Packaging Conveyor Box in Position"
  I:0.4  "Spare Analog Input 1"
  I:0.5  "Spare Analog Input 2"
  I:0.6  "Spare Analog Input 3"
  L13:31  "do not use"
  L13:32  "do not use"
  L14:0  TESTING_ENABLED
  L14:1  BOXING_CONNECTED_OLD
  L14:2  REAR_EMERG_STOP_OLD
  L14:3  FRONT_EMERG_STOP_OLD
  L14:4  REAR_DOOR_SW_OLD
  L14:5  FRONT_DOOR_SW_OLD
  L14:6  FEED_STATUS_OLD
  L14:7  CONVEYOR_STATUS_OLD
  L14:8  POWER_STATUS_OLD
  L14:9  BOX_JAM_FAULT_OLD
  L14:10  NO_BOX_FAULT_OLD
  L14:11  DSCRG_BACKUP_FAULT
  L14:12  MACHINE_FAULT_OLD
  L14:13  CNTER_SEOR_FLT
  L14:14  TOP_CONVEY_FLT_OLD
  L14:15  DN_TRACK_BLOD_FLT
  L14:16  AIR_PRESSURE_FAULT_O
  L14:17  AIR_PRESSURE_OLD
  L14:18  AIR_PRESSUREB
  L14:19  CURRENT_BOX_COUNT
  L14:20  CURRENT_BOX_COUNTB
  L14:21  PASSING_PART_COUNT
  L14:22  PASSING_PART_COUNTB
  L14:24  FAILING_PART_COUNTB
  L14:25  RATE
  L14:26  RATEB
  L14:27  RATE_DROP
  L14:28  RATE_DROPB
  L14:29  NON_PASS_BOT
  L14:30  NON_PASS_BOTB
  L14:31  NON_PASS_SIDE
  L14:32  NON_PASS_SIDEB
  L14:33  NON_PASS_TOP
  L14:34  NON_PASS_TOPB
  L14:35  CAM_NON_PASS
  L14:36  CAM_NON_PASSB
  L14:37  TOP_OPT_FAIL_CT_OLD
  L14:38  TOP_OPT_FAIL_CTB
  L14:39  BOT_OPT_FAIL_CT_OLD
  L14:40  BOT_OPT_FAIL_CTB
  L14:41  OPTO_FAILS
  L14:42  OPTO_FAILSB
  L14:43  TOO_CLOSE_BOT_OLD
  L14:44  TOO_CLOSE_BOTB
  L14:45  TOO_WIDE_BOT_OLD
  L14:46  TOO_WIDE_BOTB
  L14:47  ALIGN_FAILS_OLD
  L14:48  ALIGN_FAILSB
  L14:49  TOO_CLOSE_TOP_OLD
  L14:50  TOO_CLOSE_TOPB
  L14:51  TOO_WIDE_TOP_OLD
  L14:52  TOO_WIDE_TOPB
  L14:53  I1_REJECTS_FLT
  L14:54  FEED_WHEEL_STATUS
  L14:55  I2_REJECTS_FLT
  L14:56  I3_REJECTS_FLT
  L14:57  TOP_OP_REJECTS_FLT_O
  L14:58  BOT_CONVEY_FLT_OLD
  L14:59  BOTTOTOPALIGNMENT_OL  "Measurement of last offset of part alignment for part tracking between bottom system & top"
  L14:60  BOTTOTOPALIGNMENTB  "Measurement of last offset of part alignment for part tracking between bottom system & top"
  L14:61  TOP_BELT_SPEED_OLD  "Top Belt Speed x 1000"
  L14:62  TOP_BELT_SPEEDB  "Top Belt Speed B x 1000"
  L14:63  BOT_BELT_SPEED_OLD  "Bot Belt Speed x 1000"
  L14:64  BOT_BELT_SPEEDB  "Bot Belt Speed B x 1000"
  L14:65  BULK_DONE
  L15:0  MAX_PART_WIDTH_BOT_O
  L15:1  NU1
  L15:2  BOT_CAM_TRIG_POS
  L15:3  BOT_CAM_TRIG_POSB
  L15:4  BOT_TRANS_POINT_OLD
  L15:5  BOT_TRANS_POINTB
  L15:6  TRANS_ZONE_WIDTH_OLD
  L15:7  TRANS_ZONE_WIDTHB
  L15:8  TOP_OPTIC_POS_OLD
  L15:9  TOP_OPTIC_POSB
  L15:10  MAX_PART_WIDTH_TOP_O
  L15:11  MAX_PART_WIDTHB
  L15:12  MIN_PART_GAP_TOP_OLD
  L15:13  MIN_PART_GAP_TOPB
  L15:14  SIDE_CAM_TRIG_POS_OL
  L15:15  SIDE_CAM_TRIG_POSB
  L15:16  EXTRA_TRIG_POS
  L15:17  EXTRA_TRIG_POSB
  L15:18  TOP_CAM_TRIG_POS
  L15:19  TOP_CAM_TRIG_POSB
  L15:20  BLOW_OFF_POSITION_OL
  L15:21  BLOW_OFF_POSITIONB
  L15:22  MAX_CONT_REJECT
  L15:23  MAX_CONT_REJECTB
  L15:24  TOP_LOAD_POSITION_OL
  L15:25  TOP_LOAD_POSITIONB
  L15:26  BLOW_TIME_OLD
  L15:27  BLOW_TIMEB
  L15:28  BOT_CONV_SPEED_OLD
  L15:29  BOT_CONV_SPEEDB
  L15:30  TOP_CONV_SPEED_OLD
  L15:31  TOP_CONV_SPEEDB
  L15:32  BOX_COUNT_LIMIT_OLD
  L15:33  BOX_COUNT_LIMITB
  L15:34  BOT_OPTIC_LOC_OLD
  L15:35  BOT_OPTIC_LOCB
  L15:36  MIN_PART_GAP_BOT_OLD
  L15:37  MIN_PART_GAP_BOTB
  L15:38  FEEDER_SPEED_OLD  "15% min"
  L15:39  FEEDER_SPEEDB  "15% min"
  L15:40  HOPPER_SPEED_OLD  "15% min"
  L15:41  HOPPER_SPEEDB  "15% min"
  L15:42  ENABLE_BOXING_OLD
  L15:43  RESET_PLC_FAULT_OLD
  L15:44  ALIGNMENT_TRIGGERS_O
  L15:45  ENABLE_AIR_FAULT_OLD
  L15:46  TURN_OFF_CON_OLD  "HMI Stop Conveyors Push Button"
  L15:47  TURN_ON_CONVEYORS_OL  "HMI Start Conveyors Push Button"
  L15:48  TURN_OFF_FEEDER_OLD  "HMI Stop Feeder Push Button"
  L15:49  TURN_ON_FEEDER_OLD  "HMI Start Feeder Push Button"
  L15:50  RESET_ALL_COUNT_OLD
  L15:51  FORCE_PLC_FAULT
  L15:52  ENABLE_INSPECTION1
  L15:53  ENABLE_INSPECTION2_O
  L15:54  ENABLE_INSPECTION3
  L15:55  ENABLE_INSPECTION4
  L15:56  VISION_MAX_RES_MS_OL
  L15:57  VISION_MAX_RES_MSB
  L15:58  VISION_MIN_RES_MS
  L15:59  VISION_MIN_RES_MSB
  L15:60  RESET_FAIL_COUNT_OLD
  L15:61  RESET_BOX_COUNT_OLD  "HMI Box count Reset"
  L15:62  FEED_WHEEL_START
  L15:63  FEED_WHEEL_STOP
  L15:64  FEED_WHEEL_SPEEDOLD
  L15:65  FEED_WHEEL_SPEEDB
  L15:66  MAX_BLOW2CHUTE_MS_OL
  L15:67  MAX_BLOW2CHUTE_MSB
  L15:68  BULK_ENABLE
  L23:48  RATE_LAST_PPM
  L23:54  MAXRATEDROP_FAULT
  L24:5  ENABLE_BOXING
  L24:50  MAXDROP
  L24:53  SETUP_REQUEST
  N7:28  BOT_TRIG_POS_OLD  "Trigger Position"
  N7:38  "blow to optic time"
  N7:41  "Maximum Time from blow Signal to Optic Chute Optic Crosing MAX_BLOW2CHUTE_MS"
  N7:44  LAST_BOT_OFFSET_R  "Last part offset since pass from trigger location for setup evaluation"
  N7:45  SIDE_TEST_WIDTH  "side pass zone width"
  N7:51  "side camera response time ms"
  N7:52  "Part Rate as interger"
  N7:53  "bot belt speed as interger"
  N7:54  "side camera responce distance"
  N7:55  "top camera responce distance"
  N7:56  "top camera responce time ms"
  N7:63  "min part spacing bottom"
  N7:77  BOT_TEST_WIDTH  "bot pass zone width"
  N7:79  "bottom top camera responce distance"
  N7:80  "bottom top camera responce time"
  N7:81  "bottom to top offset"
  N7:83  "last part count for rate"
  N7:85  "measure movement"
  N7:86  "fake part optic far edge position to virtual real part"
  N7:101  3ED_BOT
  N7:103  3ED_SIDE
  N7:105  3ED_TOP
  N10:1  "old ConveyorStatus"
  N10:2  "PowerOn"
  N10:3  "Local Mode On BypassBoxingPLC"
  N10:4  "Boxing Connected Signal"
  N10:5  "BoxJamSignal"
  N10:6  "WaittingOnBoxSig"
  N10:7  "ConveyorFullSig"
  N10:8  "MachineFaultSig"
  N10:9  "Counter Sensor Fault"
  N10:11  "Feeder Track Sensor Blocked"
  N10:12  "Air Pressure Fault"
  N13:0  "Part Inspecting"
  N13:4  "Completed Counter"
  N13:5  "Trigger Position Counter"
  N13:6  "BlowOff Start Counter"
  N13:7  "BlowOff Stop Counter"
  N13:8  "Inspection Command Counter"
  N13:9  "Complete Counter"
  N13:10  "Pass Signal Counter"
  N13:11  "Solenoid Signal Counter"
  N13:12  "Hold Pass Counter"
  N13:13  "Hold Pass Length"
  N16:0  BOT_TRIGGER_OLD  "Trigger Position"
  N16:1  "Bottom Inspection Offset For Tracking"
  N16:3  "Bit Shift Preset"
  N17:5  "Parts In Tube Counter"
  N17:6  "Parts In Tube Limit"
  N17:9  "Bot to Top Transfer Position"
  N17:12  "Trigger to laser Counter"
  O:0.0/1  TOP_RINGLIGHT  "Camera "F" Top View Ringlight Enable"
  O:0.0/6  "Spare"
  O:0.0/11  "Spare"
  O:0.5  SPARE_ANALOG  "Spare analog signal"
  OUR  
  PFILE:6  "check for part jams"
  PFILE:26  "Justin's customer bo xer ladder"
  R6:5.POS  "Empty Fifo"
  R21:0  "Trigger Shift Register"
  T4:32  "Boxing Signal Conveyor Moving Debounce Bit"
  T4:33  "Packaging Good Oneshot Timer"
  T20:0  "Trigger On Time"
  T23:0  T25
  U:31  "rate calc"
  U:34  "customer boxing unit signals"

OTHER INSTRUCTION COMMENTS
  ENABLE_I1 XIC  "ENABLE_I1"

COMMENTS NOT ATTACHED TO A CURRENT RUNG
  F8:13: *************************
    Loads Side Camera Passing data into a bit shift
    *************************
    
    loads passing data bit into passing data bit shift register at the part present cl.
  I:0.0/8: special rung for testing. This rung can simulate a pass signal. It will not be timed correctly.
  B23:0/0: Yet another bit shift load with data in the part position indicating that there was a bottom system part pass as well as a top system part present at this location.
    
    verified works w/bypassed 071910 and unbypassed 072010
  N7:25: 1050
  C5:4: tempory counting to verify pass part count with boxing part count.
  B22:0/0: ***********************
     Bottom Part Syncronizing Logic
    ***********************
    
    This is the point at the bottom of the top conveyor where the part jumps from the bottom conveyor.  This system will then track the part through the top system to the point of the laser optic in order to verify that the part in question has passed the bottom inspection.  I believe that we NEED to include FAILING inspections to eliminate the possibility of a out of position part from passing. LW 072010
  T20:2.ACC: This rung is starting a timer that should be activated directly before the laser optic part presense sensor on the top conveyer and should cause the top optic to be ignored if the bottom camera system didn't pass. however other arrangements must be made if the bottom camera isn't going to be used as is the case with a nut inspection.
  T20:2: The timer used to verify that the part that triggered the top laser optic has passed the bottom camer. needs to be count
  N17:8: ****************************************************************************************************************
    I can not find anywhere in the program where the "Test Spacing From Pickup to Trigger is activated indicating to me that this entire function must not be doing anything in this program at this time.
    ****************************************************************************************************************
  B11:0/0: load part present bit shit with one shot data from the part present sensor
  B3:7/9: ************************************
     The next 3 rungs appear to do nothing
    ***********************************
  T4:0: **************
    Side Camera Trigger
    *************
    
    Trigger top camera (side)
  B3:6/0: make a bit come on indicating that a part that passed the bottom camera is within  range when crossing the top camera.
  F8:0: Counter inside of a high speed counter interrupt counts the number of Bit Shifts that need to be processed in order to move the logic with the parts on the conveyor.
  N7:45: not fully functional because of part overlap but measurems the camera responce time when part inspections are not overlaping
  B3:0/7: ********************
    Passing Part at Blow Position
    
    Blow signal is not retriggerable. If any signals are received prior to previous compleation of the blow process the signal will be ignored. Future changes may include tests or faults to verify that multiple blow signals are not overlaping.
    ********************
  O:0.0/3: **************
    Side Camera Trigger
    *************
  B9:0/[N7:47]: Remove any part present signals outside of expected location
  O:0.0/2: **************
    Side Camera Trigger
    *************
  B9:0/[N7:50]: Remove any part present signals outside of expected location
  F19:0: Counter inside of a high speed counter interrupt counts the number of Bit Shifts that need to be processed in order to move the logic with the parts on the conveyor.
  B3:4/14: *****
    Convertion of the optic signal to something stable
    *****
  F8:14: **************
    Bottom Top Camera Trigger
    *************
    
    Trigger Bottom Top Camera
  N10:4: test if boxing is connected
  B3:6/8: ********************************************************************************************************************************
    Box count reached
    Redo all of boxing;
    1. handle box done, change, box not moving, no new box
    2. everything else is situational, i.e. box removed, box not present
    add bulk pack rutine that just stops bowl and doesn't change box.
    ********************************************************************************************************************************
  T4:27: Time to clear shoot
  B3:6/9: Detect fault condition no box present on conveyor
  L13:2: Reset box count
  T4:28: Time to close shoot door
  L13:20: The following lines of code calculate the minimum and maximum time between evaluations. This is used for troubleshooting result timing issues.
  L14:8: on when ok for run
  L14:3: off when ok to run
  L14:2: off when ok to run
  L14:5: on when ok to run, rear off turns both off
  N7:76: removed relieance on trigger signal
  L14:23: ****************  nEEDS fIXING  **********************
  L14:36: ****************  nEEDS fIXING  **********************

REVISION NOTES
  13: updated count reset
  14: added io moduals
  15: multiple steps toward new hmi integration
  21: test

DATA TABLE (non-zero values as saved)
DATA B3
% B3:0 % 0X701C 0X0026 0X0000 0X0626 0X0C4A 0X6400 0X02C0 0X0020 0X0017 0X1020
% B3:10 % 0X2043 0X0846 0X2000 0X4004 0X8005
DATA T4
% .PRE .ACC %
% T4:0 % 12 0
% T4:1 % 12 0
% T4:2 % 10000 0
% T4:3 % 5 5
% T4:4 % 8 0
% T4:5 % 35 35
% T4:6 % 3 3
% T4:7 % 12 0
% T4:8 % 300 0
% T4:9 % 30 0
% T4:10 % 35 35
% T4:11 % 500 192
% T4:12 % 50 0
% T4:13 % 999 0
% T4:14 % 333 0
% T4:15 % 180 0
% T4:16 % 999 0
% T4:17 % 300 0
% T4:18 % 8 0
% T4:19 % 6 0
% T4:20 % 8 0
% T4:21 % 100 0
% T4:22 % 20 20
% T4:23 % 900 0
% T4:24 % 120 0
% T4:25 % 250 0
% T4:26 % 666 666
% T4:27 % 400 0
% T4:29 % 100 0
% T4:30 % 50 0
% T4:31 % 20 20
% T4:32 % 2 2
% T4:33 % 5 5
% T4:34 % 1000 0
% T4:35 % 22 0
% T4:36 % 1000 1003
DATA R6
% .LEN .POS %
% R6:0 % 2000 0
% R6:1 % 600 0
% R6:2 % 2000 0
% R6:4 % 1600 0
% R6:6 % 1600 0
DATA N7
% N7:0 % 1238 46 20 0 66 127 1503 45 45 32767
% N7:10 % 6 5 1239 57 1499 121 40 1042 60 39
% N7:20 % 5 120 57 10 0 30 -390 30 132 650
% N7:30 % 30 1007 1002 256 652 32767 16 9 0 0
% N7:40 % 1186 180 1247 1498 9 0 32767 1295 1246 32767
% N7:50 % 1303 0 175 16 0 0 0 1501 5 0
% N7:60 % 1 32767 66 20 76 41 256 15 30 20
% N7:70 % 0 21 23 0 32767 57 177 0 16 0
% N7:80 % 0 6 100 0 0 0 5 0 0 0
% N7:90 % 2011 4 4 12 1 0 0 0 0 1600
% N7:100 % 178 145 1296 1234 1304 1239 0 2239 0 0
% N7:110 % 0 0 0 0 0 0 0 0 50 0
% N7:120 % 25007 0 0 0 0 0 0 0 0 0
DATA F8
% F8:0 % 0.4040115 222 44928.89 44939.67 0
% F8:10 % 44.93967 0.08897486 1243 0.06033325 44.92889
% F8:15 % 0.07110977 0.3016663 51.2 256.7981 51.2
% F8:20 % 256.5892 0.02 0 0 0
% F8:25 % 0.4844475 932781 0.222 279.6551 4317
% F8:30 % 0 170 0.03 38 852060
% F8:35 % 0 0 0 0 77
% F8:40 % 0.158268 0.0968895 0 100 1
% F8:45 % 1 2 0.21455 0 0
% F8:50 % 0 0 1 0 1
% F8:55 % 0 -221 0 0 0
DATA B9
% B9:130 % 0X0000 0X0000 0X0000 0X0000 0X2000 0X0000 0X0000 0X0000 0X0000 0X8000
% B9:140 % 0X2480 0X0000 0X0000 0X0000 0X0000 0X0000 0X0000 0X0000 0X0000 0X0000
% B9:160 % 0X0000 0X0000 0X0000 0X0000 0X0000 0X0000 0X2000 0X0002 0X0000 0X0000
% B9:170 % 0X0000 0X0000 0X0000 0X2000 0X0000 0X0000 0X0000 0X0000 0X0000 0X0000
% B9:180 % 0X0000 0X0000 0X0000 0X0000 0X0000 0X0002 0X0000 0X0000 0X0000 0X0000
% B9:190 % 0X0010 0X0000 0X0000 0X0000 0X0000 0X0000 0X0000 0X0000 0X0000 0X0000
% B9:200 % 0X2B64 0X2B64 0X0000 0X0010 0X0000 0X2000 0X0000 0X0000 0X0000 0X0000
% B9:220 % 0X0000 0X0000 0X0000 0X0200 0X0000 0X0000 0X0000 0X0000 0X0000 0X0020
% B9:230 % 0X0040 0X0000 0X0000 0X0000 0X0000 0X0000 0X0000 0X0000 0X0000 0X0000
DATA B11
% B11:180 % 0X0000 0X8000 0X0000 0X0000 0X0000 0X0000 0X0000 0X0000 0X0000 0X0000
% B11:240 % 0X0000 0X0000 0X0000 0X4000 0X0000 0X0000 0X0000 0X0000 0X0000 0X0000
DATA L13
% L13:0 % 10000 0 141 85 1034016926
% L13:5 % 50 350 1000000 1034016922 1034016995
% L13:10 % 68 174024767 349654755 14368722 14368689
% L13:15 % 859992159 65535 -65536 2147483647 89612550
% L13:20 % 27597 860000727 10252744 947 2785
% L13:25 % 32767 1034025524 174024720 860000804 3125
% L13:30 % 280 200000 500000 4 32767
% L13:35 % 225 225 225 0 32767
% L13:40 % 1 0 28 14368621 3832
% L13:50 % -2147483648 2147483647 2147483647 0 0
DATA L23
% L23:0 % 65535 65535 -65536 -65536 65535
% L23:5 % 65535 65535 110 65535 65535
% L23:10 % -65536 0 0 12 0
% L23:20 % 0 -65536 -65536 -65536 -65536
% L23:25 % -65536 8 4 4 85
% L23:30 % 56 0 -65536 -65536 -65536
% L23:35 % -65536 -65536 -65536 -65536 -65536
% L23:40 % 12143 12878 45087 45063 65535
% L23:45 % 208 0 0 0 0
% L23:50 % 0 -65536 -65536 141 -65536
% L23:55 % 4040 349 -65536 8 8
% L23:60 % 8 -65536 65535 -65536 -65536
% L23:65 % -65536 0 0 0 0
DATA L24
% L24:0 % -65536 120 -65536 999 -65536
% L24:5 % 65535 -65536 -65536 -65536 -65536
% L24:10 % 76 22 60 1 23
% L24:15 % 1186 1002 100 16 20
% L24:20 % 30 -65536 1238 65535 -65536
% L24:25 % 333 1246 65535 -65536 999
% L24:30 % 1503 50 20 -65536 55
% L24:35 % 180 -65536 180 65535 45
% L24:40 % 45 5 -65536 -65536 10
% L24:45 % 222 192 -65536 3 -65536
% L24:50 % -999 30 10000 65535 900
% L24:55 % 400 65535 0 0 0
DATA L42
% L42:0 % -65536 0 0 0 0
% L42:5 % 45 45 45 0 0
% L42:20 % 0 0 32766 32766 0
% L42:30 % 0 0 97 0 0
% L42:50 % 0 30
